{attribute 'linkalways'} 
{attribute 'no_explicit_call' := 'This FB is a CLASS and must be accessed using methods or properties'}
{attribute 'enable_dynamic_creation'}
FUNCTION_BLOCK _BYTE EXTENDS NumericDatatypeBase IMPLEMENTS I_BYTE
VAR
	localData : BYTE;
	activeData : REFERENCE TO BYTE REF= localData;
END_VAR

PROPERTY PUBLIC Address : PVOID
GET
Address := ADR(activeData);
END_GET
END_PROPERTY

METHOD PUBLIC ClearReference
VAR_INPUT
END_VAR
activeData REF= localData;
END_METHOD

METHOD PUBLIC Clone : I_Datatype
VAR
    pClone : POINTER TO _BYTE;
END_VAR
pClone := __NEW(_BYTE(InitialValue := Value));
Clone := pClone^;
END_METHOD

METHOD FB_init : BOOL
VAR_INPUT
	bInitRetains : BOOL; // if TRUE, the retain variables are initialized (warm start / cold start)
	bInCopyCode : BOOL;  // if TRUE, the instance afterwards gets moved into the copy code (online change)
	InitialValue : BYTE;
END_VAR
localData := InitialValue;
END_METHOD

PROPERTY PUBLIC IsEven : BOOL
GET
IsEven := (Value mod 2) = 0;
END_GET
END_PROPERTY

PROPERTY PUBLIC IsFloat : BOOL
GET
IsFloat := FALSE;
END_GET
END_PROPERTY

PROPERTY PUBLIC IsSigned : BOOL
GET
IsSigned := FALSE;
END_GET
END_PROPERTY

METHOD PUBLIC MakeReferenceTo
VAR_INPUT
	ReferenceTarget : REFERENCE TO BYTE;
END_VAR
activeData REF= ReferenceTarget;
END_METHOD

PROPERTY PUBLIC MaxValue : BYTE
GET
MaxValue := DatatypeLimits.BYTE_MAX_VALUE;
END_GET
END_PROPERTY

PROPERTY PUBLIC MinValue : BYTE
GET
MinValue := DatatypeLimits.BYTE_MIN_VALUE;
END_GET
END_PROPERTY

METHOD PROTECTED SerializeMaxValue
VAR_INPUT
	Serializer : I_Serializer;
END_VAR
Serializer.AddByte(MaxValue);
END_METHOD

METHOD PROTECTED SerializeMinValue
VAR_INPUT
	Serializer : I_Serializer;
END_VAR
Serializer.AddByte(MinValue);
END_METHOD

METHOD PUBLIC SerializeWith
VAR_INPUT
	Serializer : I_Serializer;
END_VAR
Serializer.AddByte(activeData);
END_METHOD

PROPERTY PUBLIC Size : UDINT
GET
Size := SIZEOF(activeData);
END_GET
END_PROPERTY

METHOD PUBLIC TryConvertTo : BOOL
VAR_INPUT
	Destination : ANY;
END_VAR
TryConvertTo := TryConvert_BYTE_To_Destination(activeData, Destination);
END_METHOD

METHOD PUBLIC TryConvertTo_ : BOOL
VAR_INPUT
	Destination : I_Datatype;
END_VAR
VAR
	resultofBitConversion : BOOL;
	destinationAs_BIT : I_BIT;
	destinationAs_BOOL : I_BOOL;
	destinationAs_BYTE : I_BYTE;
	destinationAs_DINT : I_DINT;
	destinationAs_DT : I_DT;
	destinationAs_DWORD : I_DWORD;
	destinationAs_INT : I_INT;
	destinationAs_LINT : I_LINT;
	destinationAs_LREAL : I_LREAL;
	destinationAs_LWORD : I_LWORD;
	destinationAs_REAL : I_REAL;
	destinationAs_SINT : I_SINT;
	destinationAs_STRING : I_STRING;
	destinationAs_TOD : I_TOD;
	destinationAs_UDINT : I_UDINT;
	destinationAs_UINT : I_UINT;
	destinationAs_ULINT : I_ULINT;
	destinationAs_USINT : I_USINT;
	destinationAs_WORD : I_WORD;
END_VAR
IF destination.TryResolveAs_BIT(destinationAs_BIT) AND_THEN TryConvert_BYTE_TO_BOOL(activeData, resultofBitConversion) THEN
	destinationAs_BIT.Value := resultOfBitConversion;
	TryConvertTo_ := TRUE;
	RETURN;
END_IF

IF destination.TryResolveAs_BOOL(destinationAs_BOOL) THEN
	TryConvertTo_ := TryConvert_BYTE_TO_BOOL(activeData, destinationAs_BOOL.Value);
	RETURN;
END_IF
		
IF destination.TryResolveAs_BYTE(destinationAs_BYTE) THEN
	TryConvertTo_ := TryConvert_BYTE_TO_BYTE(activeData, destinationAs_BYTE.Value);
	RETURN;
END_IF

IF destination.TryResolveAs_DINT(destinationAs_DINT) THEN
	TryConvertTo_ := TryConvert_BYTE_TO_DINT(activeData, destinationAs_DINT.Value);
	RETURN;
END_IF

IF destination.TryResolveAs_DT(destinationAs_DT) THEN
	TryConvertTo_ := TryConvert_BYTE_TO_DT(activeData, destinationAs_DT.Value);
	RETURN;
END_IF

IF destination.TryResolveAs_DWORD(destinationAs_DWORD) THEN
	TryConvertTo_ := TryConvert_BYTE_TO_DWORD(activeData, destinationAs_DWORD.Value);
	RETURN;
END_IF

IF destination.TryResolveAs_INT(destinationAs_INT) THEN
	TryConvertTo_ := TryConvert_BYTE_TO_INT(activeData, destinationAs_INT.Value);
	RETURN;
END_IF

IF destination.TryResolveAs_LINT(destinationAs_LINT) THEN
	TryConvertTo_ := TryConvert_BYTE_TO_LINT(activeData, destinationAs_LINT.Value);
	RETURN;
END_IF

IF destination.TryResolveAs_LREAL(destinationAs_LREAL) THEN
	TryConvertTo_ := TryConvert_BYTE_TO_LREAL(activeData, destinationAs_LREAL.Value);
	RETURN;
END_IF

IF destination.TryResolveAs_LWORD(destinationAs_LWORD) THEN
	TryConvertTo_ := TryConvert_BYTE_TO_LWORD(activeData, destinationAs_LWORD.Value);
	RETURN;
END_IF

IF destination.TryResolveAs_REAL(destinationAs_REAL) THEN
	TryConvertTo_ := TryConvert_BYTE_TO_REAL(activeData, destinationAs_REAL.Value);
	RETURN;
END_IF

IF destination.TryResolveAs_SINT(destinationAs_SINT) THEN
	TryConvertTo_ := TryConvert_BYTE_TO_SINT(activeData, destinationAs_SINT.Value);
	RETURN;
END_IF

IF destination.TryResolveAs_STRING(destinationAs_STRING) THEN
	TryConvertTo_ := TryConvert_BYTE_TO_STRING(activeData, destinationAs_STRING.Value);
	RETURN;
END_IF

IF destination.TryResolveAs_TOD(destinationAs_TOD) THEN
	TryConvertTo_ := TryConvert_BYTE_TO_TOD(activeData, destinationAs_TOD.Value);
	RETURN;
END_IF

IF destination.TryResolveAs_UDINT(destinationAs_UDINT) THEN
	TryConvertTo_ := TryConvert_BYTE_TO_UDINT(activeData, destinationAs_UDINT.Value);
	RETURN;
END_IF

IF destination.TryResolveAs_UINT(destinationAs_UINT) THEN
	TryConvertTo_ := TryConvert_BYTE_TO_UINT(activeData, destinationAs_UINT.Value);
	RETURN;
END_IF

IF destination.TryResolveAs_ULINT(destinationAs_ULINT) THEN
	TryConvertTo_ := TryConvert_BYTE_TO_ULINT(activeData, destinationAs_ULINT.Value);
	RETURN;
END_IF

IF destination.TryResolveAs_USINT(destinationAs_USINT) THEN
	TryConvertTo_ := TryConvert_BYTE_TO_USINT(activeData, destinationAs_USINT.Value);
	RETURN;
END_IF

IF destination.TryResolveAs_WORD(destinationAs_WORD) THEN
	TryConvertTo_ := TryConvert_BYTE_TO_WORD(activeData, destinationAs_WORD.Value);
	RETURN;
END_IF
END_METHOD

METHOD TryDeserializeFrom : BOOL
VAR_INPUT
	Deserializer : I_Deserializer;
	Feedback : I_DeserializerFeedback;
END_VAR
TryDeserializeFrom := Deserializer.TryGetByte(activeData, Feedback);
END_METHOD

METHOD TryMakeReferenceTo : BOOL
VAR_INPUT
	Target : I_Datatype;
END_VAR
VAR
	pTargetData : POINTER TO BYTE;
END_VAR
IF NOT IsEquivalentTo(Target) THEN
	RETURN;
END_IF

pTargetData := Target.Address;
activeData REF= pTargetData^;
TryMakeReferenceTo := TRUE;
END_METHOD

METHOD PUBLIC TryResolveAs_BYTE : BOOL
VAR_INPUT
	Destination : REFERENCE TO I_BYTE;
END_VAR
Destination := THIS^;
TryResolveAs_BYTE := TRUE;
END_METHOD

PROPERTY PUBLIC TypeName : T_MAXSTRING
GET
TypeName := 'BYTE';
END_GET
END_PROPERTY

PROPERTY PUBLIC Value : REFERENCE TO BYTE
GET
Value REF= activeData;
END_GET
END_PROPERTY

END_FUNCTION_BLOCK

(* stored: Version 1.1.0.1, ProductVersion 3.1.4024.15
   POU _BYTE: Id {015fee84-30df-4efb-96c8-fa65eaa5aa83}, SpecialFunc None
   Folder Constructor: Id {52a26577-a6bc-4aa5-9ef8-f187627d1642}
   Folder Protected: Id {8aa9057a-15bb-4079-bf78-cfd21590127a}
   Property Address: Id {f4658331-4fdd-43d9-be9e-00542c59946a}
   Get Get: Id {d753ed97-43be-40c2-a48d-d6d299103d65}
   Method ClearReference: Id {3854d391-b7b2-4b47-9f9a-18e69b0dcbda}
   Method Clone: Id {e218fd2c-90c0-45b2-a3dc-c3ce9829dc9a}
   Method FB_init: Id {c73f40e7-da83-43bf-b9c3-680c5d3df281}
   Property IsEven: Id {0bd65d0c-d483-08a8-3b31-f7c1093a4208}
   Get Get: Id {65b92a46-be93-0abd-3c3f-3f58d52dd0fb}
   Property IsFloat: Id {65b20559-d076-483f-b3d3-9f65fcb52652}
   Get Get: Id {e8ca72cd-2c65-4183-94e9-64387bc9c4f2}
   Property IsSigned: Id {83a3b0ce-180f-4907-989b-f922d0f2214e}
   Get Get: Id {d6690cbf-d958-4d50-9841-8375714a31ff}
   Method MakeReferenceTo: Id {18ec47ae-83dd-4afc-a3f0-890a89595ae0}
   Property MaxValue: Id {47ded2cf-bef0-4212-afe1-d53ae7a8073a}
   Get Get: Id {be9751fc-c4c7-4b02-b040-d761b9f03f84}
   Property MinValue: Id {b0a5acb4-937e-49e0-ae6b-7185073a6fe6}
   Get Get: Id {8b359cfc-8c76-478a-a1b9-a2dfcc7188e4}
   Method SerializeMaxValue: Id {2b2dd19b-d33d-47a5-a3fd-8f7871724ec3}
   Method SerializeMinValue: Id {6bd0c9eb-7393-4705-994d-fa6038d95d76}
   Method SerializeWith: Id {66fb1589-93aa-48cc-9b7f-87181c23e74d}
   Property Size: Id {7f95387a-676f-4254-8a17-a3b6e9673cda}
   Get Get: Id {128d205a-ce0d-44fe-9ee1-7b8137c3ed50}
   Method TryConvertTo: Id {981a87df-021f-0aa1-395a-035f336848f6}
   Method TryConvertTo_: Id {16ef359b-d366-0efd-091a-3e78877caf79}
   Method TryDeserializeFrom: Id {ed654a62-7512-4173-bcd9-55f451d1c2af}
   Method TryMakeReferenceTo: Id {dc7c26da-384c-431a-824b-f41d2d332124}
   Method TryResolveAs_BYTE: Id {4bae1ce9-09a6-0fc1-0632-bc5ce64b6e7e}
   Property TypeName: Id {1c1c2320-0402-4c90-bee9-948e0946fa55}
   Get Get: Id {2f3ac17e-d722-4c9a-a69e-7923adb5d499}
   Property Value: Id {2e144ab6-c08f-45e7-82aa-2cda5774589e}
   Get Get: Id {43823d97-4013-4032-a00f-d395ded07007} *)
